PROGRAM MAIN
VAR
	s_ParamPathnames : ARRAY[1..Param_Project.n_MaxParamFolders] OF STRING := ['C:\Cleanroom_Connect\Parameters'];
	
	User : STRING := '<user_name>';
	SoftwareVersion : STRING := '<software_version>';
	InitDone : BOOL;
	Shutdown : BOOL;
	
	fbModeStateControl : FB_ModeStateControl;
END_VAR

GVL_KMWEGenericLib.g_fbAlarmManager();

GVL_KMWEGenericLib.g_fbParamManager.p_bShowHmiParam := TRUE;

GVL_KMWEGenericLib.g_fbParamManager(
	i_sPathName := s_ParamPathnames,
	i_osrResetImportExport := GVL_KMWEGenericLib.g_fbAlarmManager.p_osrReset);

fbModeStateControl();

GVL.g_unCleanroomConnect.p_bCmdReset := GVL_KMWEGenericLib.g_fbAlarmManager.p_osrReset;
GVL.g_unCleanroomConnect();

END_PROGRAM

(* stored: Version 1.1.0.1, ProductVersion 3.1.4024.12
   POU MAIN: Id {c137dca6-2078-4081-8260-8d6099001278}, SpecialFunc None *)
